PROGRAM MAIN
VAR
END_VAR

END_PROGRAM

(* stored: Version 1.1.0.1
   POU MAIN: Id {fc58933e-47a6-4fd8-a367-fd7f6c32aed5} *)
